FUNCTION REAL_TO_WORD_SAFE : WORD
VAR_INPUT
	Value: REAL;
END_VAR
VAR
END_VAR

REAL_TO_WORD_SAFE := TO_WORD(TO_INT(Value));

END_FUNCTION

(* stored: Version 1.1.0.1, ProductVersion 3.1.4024.6
   POU REAL_TO_WORD_SAFE: Id {9bd2be92-9716-41c3-8bd4-09fc3b43d50b}, SpecialFunc None *)
